{attribute 'GeneratedUsingTerminal: EL2521-0000-1016'}
{attribute addProperty BoxType "EL2521-0000-1016"}
{attribute addProperty Id "Frequency_selectAT %Q*BOOL1Disable_rampAT %Q*BOOL1Go_counterAT %Q*BOOL1Frequency_valueAT %Q*UINT2"}
{attribute addProperty CRC "959139118"}
{attribute addProperty Size "5"}
TYPE PTO_Control_392B4D2E EXTENDS OutputBase_10CEE7DE :
STRUCT
	{attribute addProperty Name "Frequency_select"}
	Frequency_select AT %Q* : BOOL;
	{attribute addProperty Name "Disable_ramp"}
	Disable_ramp AT %Q* : BOOL;
	{attribute addProperty Name "Go_counter"}
	Go_counter AT %Q* : BOOL;
	{attribute addProperty Name "Frequency_value"}
	Frequency_value AT %Q* : UINT;
END_STRUCT
END_TYPE

(* stored: Version 1.2.0.0, ProductVersion 3.1.4024.9
   DUT PTO_Control_392B4D2E: Id {e4dde0dc-8237-4391-8bd8-7d150bb488b9} *)
